{attribute 'linkalways'} 
{attribute 'no_explicit_call' := 'This FB is a CLASS and must be accessed using methods or properties'}
{attribute 'enable_dynamic_creation'}
FUNCTION_BLOCK Node_F_VN_DoubleThreshold EXTENDS VisionNode
VAR
	ipSrcImage : _ITcVnImage;
    ipDestImage : _ITcVnImage;
    fLowThreshold : _LREAL(0.0);
    fHighThreshold : _LREAL(0.0);
    fMaxValue : _LREAL(0.0);
    hrPrev : _HRESULT(S_OK);
	hresult : _HRESULT(S_OK);
END_VAR

METHOD PUBLIC  Clone : I_Node
VAR
	pNode : POINTER TO Node_F_VN_DoubleThreshold;
END_VAR
pNode := __NEW(Node_F_VN_DoubleThreshold);
Clone := pNode^;
END_METHOD

METHOD FB_init : BOOL
VAR_INPUT
	bInitRetains : BOOL; // if TRUE, the retain variables are initialized (warm start / cold start)
	bInCopyCode : BOOL;  // if TRUE, the instance afterwards gets moved into the copy code (online change)
END_VAR
AddInput('ipSrcImage', ipSrcImage);
AddParameter('fLowThreshold', fLowThreshold);
AddParameter('fHighThreshold', fHighThreshold);
AddParameter('fMaxValue', fMaxValue);
AddInput('hrPrev', hrPrev);
AddOutput('ipDestImage', ipDestImage);
AddOutput('hresult', hresult);
END_METHOD

METHOD PROTECTED OnExecute
hresult.Value := F_VN_DoubleThreshold(
	ipSrcImage := ipSrcImage.Value,
	ipDestImage := ipDestImage.Value,
    fLowThreshold := fLowThreshold.Value,
    fHighThreshold := fHighThreshold.Value,
    fMaxValue := fMaxValue.Value,
	hrPrev := hrPrev.Value);
END_METHOD

METHOD PUBLIC PreExecutionCheck
VAR_INPUT
	Check : I_PreExecutionChecks;
END_VAR
VAR
    pixelFormat : TcVnPixelFormat;
END_VAR
Check.IsTrue(ipSrcImage.IsValid, 'ipSrcImage must contain an image');
Check.IsTrue(ipSrcImage.HasChannelCount(1), 'ipSrcImage must have 1 channel');
Check.IsTrue((ipSrcImage.IsPixelDepth(8) OR
              ipSrcImage.IsPixelDepth(16) OR
              ipSrcImage.IsPixelDepth(32) OR
              ipSrcImage.IsPixelDepth(64)), 'ipSrcImage must have 8, 16, 32, or 64 bit pixel depth');

ipSrcImage.TryGetPixelFormat(pixelFormat);
Check.IsTrue(IsMaxValueCompatibleWithPixelDepth(fMaxValue.Value, pixelFormat.nElementSize), 'fMaxValue is not compatible with pixel depth');
END_METHOD

END_FUNCTION_BLOCK

(* stored: Version 1.1.0.1, ProductVersion 3.1.4024.15
   POU Node_F_VN_DoubleThreshold: Id {bd4eb3d3-8cf2-0552-26fb-2f285904c869}, SpecialFunc None
   Folder Constructor: Id {c2cc68f1-277b-0e9e-3801-d86ca7963c52}
   Method Clone: Id {a90d838b-acdc-0821-3539-cbcf9c7cd208}
   Method FB_init: Id {5b0058a3-b238-0c06-3ec6-96ec3dc5551d}
   Method OnExecute: Id {8079e562-804d-058d-1f71-3aec8167ebed}
   Method PreExecutionCheck: Id {74c44f26-109b-01c3-202f-539084748d5a} *)
